{attribute 'GeneratedUsingTerminal: EL3443-0000-0016'}
{attribute addProperty BoxType "EL3443-0000-0016"}
{attribute addProperty Id "Active_PowerAT %I*REAL4Active_EnergyAT %I*LINT8Active_Positive_EnergyAT %I*ULINT8Active_Negative_EnergyAT %I*ULINT8"}
{attribute addProperty CRC "4189363873"}
{attribute addProperty Size "28"}
TYPE Total_Active_F9B49EA1 EXTENDS InputBase_8311D824 :
STRUCT
	{attribute addProperty Name "Active_Power"}
	Active_Power AT %I* : REAL;
	{attribute addProperty Name "Active_Energy"}
	Active_Energy AT %I* : LINT;
	{attribute addProperty Name "Active_Positive_Energy"}
	Active_Positive_Energy AT %I* : ULINT;
	{attribute addProperty Name "Active_Negative_Energy"}
	Active_Negative_Energy AT %I* : ULINT;
END_STRUCT
END_TYPE

(* stored: Version 1.2.0.0, ProductVersion 3.1.4024.9
   DUT Total_Active_F9B49EA1: Id {72dc4c56-83eb-4f51-a7de-d6fe6c979281} *)
